// TwinCAT 3 PLC project _4_2_seq_autom_temporisee
// ProgramVersion: 3.1.4020.2
// libraries:
//   Tc2_Standard, * (Beckhoff Automation GmbH)
//   Tc2_System, * (Beckhoff Automation GmbH)
//   Tc3_Module, * (Beckhoff Automation GmbH)
// project tree:
//   / PlcTask.TcTTO
//   POUs/ bla.TcPOU, MAIN.TcPOU
// (motion and I/O tree: see PLC project 1calcul)
// real-time tasks:
//   TASK PlcTask: cycle T#1ms, priority 20, ADS port 350
// variable links:

CONFIGURATION _4_2_seq_autom_temporisee
    RESOURCE PLC ON TwinCAT3
        TASK PlcTask(INTERVAL := T#10ms, PRIORITY := 20);
        PROGRAM MAIN WITH PlcTask : MAIN;
    END_RESOURCE
END_CONFIGURATION

// ---- POUs/MAIN.TcPOU
PROGRAM MAIN

bla();

END_PROGRAM

// ---- POUs/bla.TcPOU
PROGRAM bla
VAR
	iStep: INT :=0; //etape
	Timer: TON;
END_VAR
VAR_INPUT
	
END_VAR
VAR_OUTPUT
	QxLED1 AT%Q* : BOOL := 0; //actionner le verin | avec AT %Q si lien physique
	QxLED2 AT%Q* : BOOL := 0; //actionner le verin | avec AT %Q si lien physique
	QxLED3 AT%Q* : BOOL := 0; //actionner le verin | avec AT %Q si lien physique
	QxLED4 AT%Q* : BOOL := 0; //actionner le verin | avec AT %Q si lien physique
END_VAR

CASE iStep OF
	0: 	Timer.PT:=T#1S;
		iStep:=100;
	100: //allumer la Lampe 1 et setter le timer 1s
			Timer.PT:=T#50MS;
			iStep:=110;
	110: //allumer la Lampe 1 et attendre 1s
		IF Timer.Q THEN
			iStep:=200;
		END_IF
	200: //allumer la Lampe 2 et setter le timer 0.5s
		Timer.PT:=T#150MS;
		iStep:=210;
	210: //allumer la Lampe 2 et attendre 0.5s
		IF Timer.Q THEN
			iStep:=300;
		END_IF
	300: //resetter LE timer
			iStep:=310;
	310: //attendre 0.5s
		IF Timer.Q THEN
			iStep:=300;
		END_IF
END_CASE
//Actions
Timer(IN:=(iStep=110 OR iStep=210 OR iStep=310));
QxLED2:=(iStep=200 OR iStep=210);
QxLED1:=(iStep=100 OR iStep=110);
QxLED3:=(iStep=200 OR iStep=210);
QxLED4:=(iStep=100 OR iStep=110);

END_PROGRAM
